(* PLC project Generated.project, CODESYS CODESYS V3.5 SP19 Patch 1 *)
(* stored: creationDateTime 2026-09-06T13:00:42.533850, modificationDateTime 2026-09-06T13:00:42.533850 *)

(* ═══════════════════════════════════════════════════════════════ 🧲 ST_AcquisitionEncoderQualified — Façade codeur qualifiée ─────────────────────────────────────────────────────────────── 🎯 Rôle : Encapsuler les mesures métriques, statuts de référencement, défauts et signaux hardware produits par FB_Encoder dans PRG_02_Acquisition. 📤 Producteur unique : PRG_02_Acquisition (Data.EncoderM1 / Data.EncoderM2). 📄 Doc : DOC/AF/AF_Partie-06_Acquisition_Qualification_IO_v2.4.md ═══════════════════════════════════════════════════════════════ *)
TYPE ST_AcquisitionEncoderQualified : STRUCT
  Measurement : ST_fbEncoder_Measurement;  (* 📊 Mesure métrique (CablePosM, SpeedMps, etc.) *)
  Ready : BOOL;  (* 🟢 Façade codeur prête *)
  Fault : ST_Fault;  (* ❌ Diagnostic défaut codeur *)
  Homed : BOOL;  (* 🎯 Codeur référencé *)
  HomingSuspect : BOOL;  (* ⚠️ Référencement suspect *)
  EncoderFault : BOOL;  (* ❌ Défaut fiabilité (indisponible ou incohérent) *)
  HomedAndReliable : BOOL;  (* ✅ Référencé ET fiable (sans incohérence) *)
  PresetConfirmationFailed : BOOL;  (* ❌ Échec confirmation preset *)
  HwOut : ST_fbEncoder_HwOut;  (* 📡 Commandes hardware de preset (lecture seule) *)
END_STRUCT;
END_TYPE

(* ======================================================================= 🧩 ST_Fault — Brique socle défaut (2 vues : live + latchée) ─────────────────────────────────────────────────────────────── 🎯 Rôle : porter l'état défaut d'un composant, applicable dans TOUS les cas (acquittable ou non), sans brique warning séparée. • Vue LIVE (Error / ErrorId) : suit la cause, retombe seule à 0. • Vue LATCHÉE (Latched / LatchedId): mémorisée au défaut, reste jusqu'au front Reset. Le choix acquittable / non-acquittable se fait PAR CAUSE (ST_FaultCause.Latching), jamais par bloc. 🔒 Sécurité : interlock TOUJOURS sur la cause brute (Error / ErrorId), jamais sur l'acquittement. Reset TOUJOURS effectif, jamais conditionné (std §9). 🧬 Composition : brique de base réutilisable — sortie de FB, struct métier, GVL. Texte IHM NON stocké ici : dérivé côté IHM depuis LatchedId / ErrorId. 📄 Doc : DOC/STDS/CODE_QUALITY_STANDARDS.md §2quinquies / §9 ======================================================================= *)
TYPE ST_Fault : STRUCT
  Error : BOOL;  (* <-- [DIAG] vue LIVE : au moins une cause présente maintenant *)
  ErrorId : WORD;  (* <-- [DIAG] bitfield des causes présentes maintenant (0 si aucune) *)
  Latched : BOOL;  (* <-- [DIAG] vue LATCHÉE : défaut non acquitté, reste jusqu'au front Reset *)
  LatchedId : WORD;  (* <-- [DIAG] ErrorId figé à l'apparition du défaut, effacé au Reset *)
END_STRUCT;
END_TYPE

(* ======================================================================= 🔌 ST_fbEncoder_HwOut — Ordres preset de sortie codeur (HwOut) ─────────────────────────────────────────────────────────────── 🎯 Rôle : Regrouper les SEULES sorties/ordres preset d'un codeur absolu EtherCAT produits par FB_Encoder vers le PDO Rx (bus sortie). 🔒 Ownership : FB_Encoder produit ce bus ; PRG_02_Acquisition le relaie vers le device. 📄 Doc métier : DOC/AF/AF_Partie-09_Fonction_Encoder_v2.4.md ======================================================================= *)
TYPE ST_fbEncoder_HwOut : STRUCT
  PresetTriggerCmd : WORD;  (* === SORTIES BUS ETHERCAT (ordres preset vers PDO Rx) === <-- [ACT] Declenchement preset vers PDO Rx *)
  CodeSeqTriggerCmd : WORD;  (* <-- [ACT] Sequence code vers PDO Rx, maintenue a 0 *)
  PresetValueOut : UDINT;  (* <-- [ACT] Valeur brute envoyee au preset *)
END_STRUCT;
END_TYPE

(* ======================================================================= 📊 ST_fbEncoder_Measurement — Mesures codeur conditionnées (1 sous-DUT par treuil) ─────────────────────────────────────────────────────────────── 🎯 Rôle : Regroupement des mesures et faits de la chaîne codeur d'un treuil (Abs → Scale → Safety → Speed) 🔌 Interface : Interface de mesure normalisée pour PRG_02_Acquisition 📄 Doc métier : DOC/AF/AF_Partie-06_Acquisition_Qualification_IO_v2.4.md ======================================================================= *)
TYPE ST_fbEncoder_Measurement : STRUCT
  RawPos : UDINT;  (* === DONNEES BRUTES & STATUT BUS === Position brute codeur (gelee si EncoderAvailable=FALSE) *)
  EncoderAvailable : BOOL;  (* TRUE = bus/esclave EtherCAT operationnel et disponible *)
  CablePosM : REAL;  (* === MESURES DE POSITION CABLE === Position cable (m, signee, + enroule) *)
  CablePosMSafe : REAL;  (* Position cable instantanee validee par EncoderIncoherent (m) *)
  EncoderIncoherent : BOOL;  (* TRUE = incoherence redemarrage ou hors bornes *)
  Speed_Mps : REAL;  (* === MESURES DE VITESSE CABLE === Vitesse absolue câble (m/s) *)
  SignedSpeed_Mps : REAL;  (* Vitesse signee câble (m/s, + montee, - descente) *)
  SpeedValid : BOOL;  (* TRUE si mesure valide et codeur operationnel *)
  HomingFault : ST_Fault;  (* === STATUTS DES SOUS-FB & REFERENCE === Défaut FB_Encoder_Homing (état du référencement) *)
  HomingLifecycle : ST_Lifecycle;  (* Cycle FB_Encoder_Homing (Busy/Done) *)
  AbsFault : ST_Fault;  (* Défaut FB_Encoder_Abs (état acquisition bus) *)
  HomingRefRaw : UDINT;  (* Reference brute du dernier homing reussi (re-expose) *)
END_STRUCT;
END_TYPE

(* ======================================================================= 🧩 ST_Lifecycle — Brique socle cycle d'exécution ─────────────────────────────────────────────────────────────── 🎯 Rôle : porter l'avancement d'une action à cycle (organe, séquenceur). Optionnelle : un FB purement synchrone (conditionneur, filtre, joystick) ne la porte pas. 🧬 Composition : brique de base réutilisable, composée avec ST_Fault. 📄 Doc : DOC/STDS/CODE_QUALITY_STANDARDS.md §2quinquies ======================================================================= *)
TYPE ST_Lifecycle : STRUCT
  Busy : BOOL;  (* <-- [STAT] 1 = action en cours *)
  Done : BOOL;  (* <-- [STAT] 1 = action terminée avec succès *)
END_STRUCT;
END_TYPE
